// TIA Portal V16 export
// export: Created 2024-06-24T15:42:27.7485025Z, ExportSetting WithDefaults, DisplayName Totally Integrated Automation Portal, DisplayVersion V16, DisplayName TIA Portal Version Control Interface, DisplayVersion V16, DisplayName TIA Portal Openness, DisplayVersion V16, DisplayName STEP 7 Professional, DisplayVersion V16, DisplayName STEP 7 Safety, DisplayVersion V16, DisplayName WinCC Advanced, DisplayVersion V16
FUNCTION_BLOCK "FB_PickAndPlace"   // FB4, LAD
{ S7_Optimized_Access := 'TRUE' }
VERSION : 0.1
// stored: AutoNumber true, IsIECCheckEnabled false, IsRetainMemResEnabled false, MemoryReserve 100, SetENOAutomatically false, UDAEnableTagReadback false
   VAR_INPUT
      machineReady : Bool;
      movingZ : Bool;
      movingX : Bool;
      itemGrabbed : Bool;
   END_VAR
   VAR_OUTPUT
      moveX : Bool;
      moveZ : Bool;
      grabItem : Bool;
   END_VAR
   VAR_IN_OUT
      start : Bool;
      done : Bool;
   END_VAR
   VAR
      "step" : Array[0..20] of Bool;
   END_VAR
   VAR_TEMP   // added for the SCL form of the ladder/FBD networks
      _w1 : Bool;
   END_VAR
BEGIN

REGION Network 1: step0
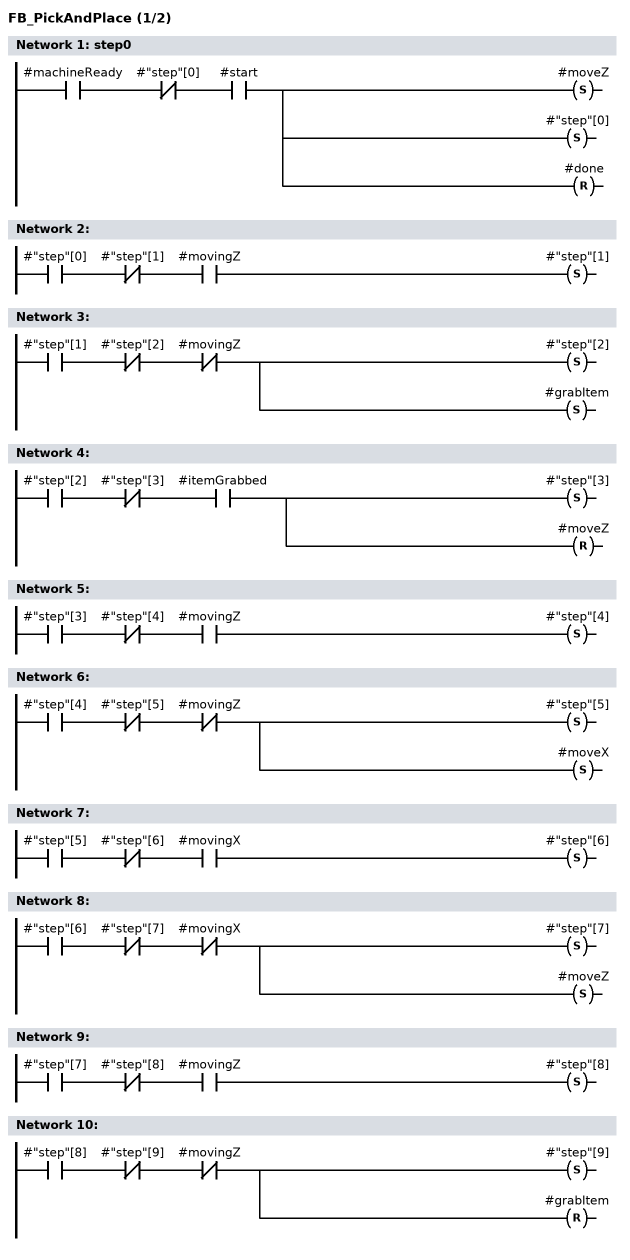
   RUNG wire#powerrail
      Contact( #machineReady )
      I_Contact( #"step"[0] )
      Contact( #start )
      wire#w1
      S_Coil( #moveZ )
   END_RUNG
   RUNG wire#w1
      S_Coil( #"step"[0] )
   END_RUNG
   RUNG wire#w1
      R_Coil( #done )
   END_RUNG
   // the same network as SCL:
   IF #machineReady AND NOT #"step"[0] AND #start THEN #moveZ := TRUE; END_IF;
   #_w1 := #machineReady AND NOT #"step"[0] AND #start;
   IF #_w1 THEN
       #"step"[0] := TRUE;
       #done := FALSE;
   END_IF;
END_REGION

REGION Network 2
   RUNG wire#powerrail
      Contact( #"step"[0] )
      I_Contact( #"step"[1] )
      Contact( #movingZ )
      S_Coil( #"step"[1] )
   END_RUNG
   // the same network as SCL:
   IF #"step"[0] AND NOT #"step"[1] AND #movingZ THEN #"step"[1] := TRUE; END_IF;
END_REGION

REGION Network 3
   RUNG wire#powerrail
      Contact( #"step"[1] )
      I_Contact( #"step"[2] )
      I_Contact( #movingZ )
      wire#w1
      S_Coil( #"step"[2] )
   END_RUNG
   RUNG wire#w1
      S_Coil( #grabItem )
   END_RUNG
   // the same network as SCL:
   #_w1 := #"step"[1] AND NOT #"step"[2] AND NOT #movingZ;
   IF #_w1 THEN
       #"step"[2] := TRUE;
       #grabItem := TRUE;
   END_IF;
END_REGION

REGION Network 4
   RUNG wire#powerrail
      Contact( #"step"[2] )
      I_Contact( #"step"[3] )
      Contact( #itemGrabbed )
      wire#w1
      S_Coil( #"step"[3] )
   END_RUNG
   RUNG wire#w1
      R_Coil( #moveZ )
   END_RUNG
   // the same network as SCL:
   #_w1 := #"step"[2] AND NOT #"step"[3] AND #itemGrabbed;
   IF #_w1 THEN
       #"step"[3] := TRUE;
       #moveZ := FALSE;
   END_IF;
END_REGION

REGION Network 5
   RUNG wire#powerrail
      Contact( #"step"[3] )
      I_Contact( #"step"[4] )
      Contact( #movingZ )
      S_Coil( #"step"[4] )
   END_RUNG
   // the same network as SCL:
   IF #"step"[3] AND NOT #"step"[4] AND #movingZ THEN #"step"[4] := TRUE; END_IF;
END_REGION

REGION Network 6
   RUNG wire#powerrail
      Contact( #"step"[4] )
      I_Contact( #"step"[5] )
      I_Contact( #movingZ )
      wire#w1
      S_Coil( #"step"[5] )
   END_RUNG
   RUNG wire#w1
      S_Coil( #moveX )
   END_RUNG
   // the same network as SCL:
   #_w1 := #"step"[4] AND NOT #"step"[5] AND NOT #movingZ;
   IF #_w1 THEN
       #"step"[5] := TRUE;
       #moveX := TRUE;
   END_IF;
END_REGION

REGION Network 7
   RUNG wire#powerrail
      Contact( #"step"[5] )
      I_Contact( #"step"[6] )
      Contact( #movingX )
      S_Coil( #"step"[6] )
   END_RUNG
   // the same network as SCL:
   IF #"step"[5] AND NOT #"step"[6] AND #movingX THEN #"step"[6] := TRUE; END_IF;
END_REGION

REGION Network 8
   RUNG wire#powerrail
      Contact( #"step"[6] )
      I_Contact( #"step"[7] )
      I_Contact( #movingX )
      wire#w1
      S_Coil( #"step"[7] )
   END_RUNG
   RUNG wire#w1
      S_Coil( #moveZ )
   END_RUNG
   // the same network as SCL:
   #_w1 := #"step"[6] AND NOT #"step"[7] AND NOT #movingX;
   IF #_w1 THEN
       #"step"[7] := TRUE;
       #moveZ := TRUE;
   END_IF;
END_REGION

REGION Network 9
   RUNG wire#powerrail
      Contact( #"step"[7] )
      I_Contact( #"step"[8] )
      Contact( #movingZ )
      S_Coil( #"step"[8] )
   END_RUNG
   // the same network as SCL:
   IF #"step"[7] AND NOT #"step"[8] AND #movingZ THEN #"step"[8] := TRUE; END_IF;
END_REGION

REGION Network 10
   RUNG wire#powerrail
      Contact( #"step"[8] )
      I_Contact( #"step"[9] )
      I_Contact( #movingZ )
      wire#w1
      S_Coil( #"step"[9] )
   END_RUNG
   RUNG wire#w1
      R_Coil( #grabItem )
   END_RUNG
   // the same network as SCL:
   #_w1 := #"step"[8] AND NOT #"step"[9] AND NOT #movingZ;
   IF #_w1 THEN
       #"step"[9] := TRUE;
       #grabItem := FALSE;
   END_IF;
END_REGION

REGION Network 11
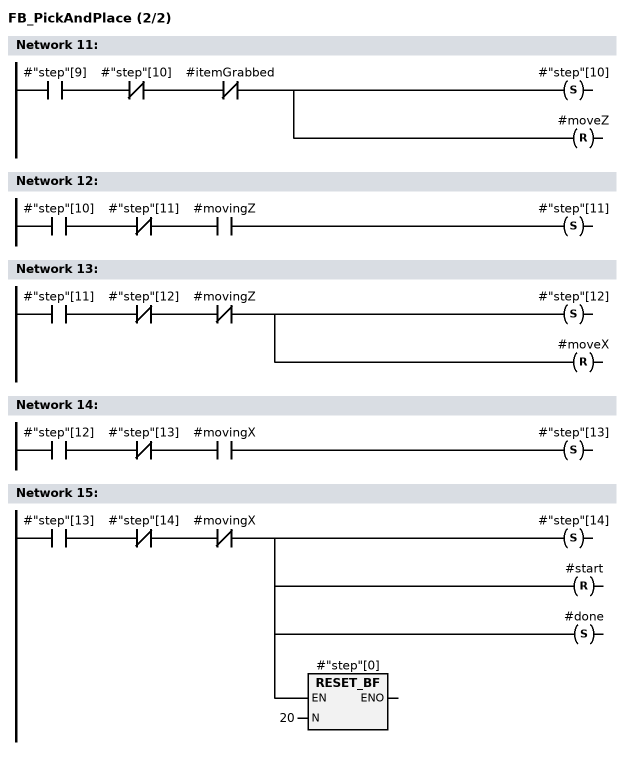
   RUNG wire#powerrail
      Contact( #"step"[9] )
      I_Contact( #"step"[10] )
      I_Contact( #itemGrabbed )
      wire#w1
      S_Coil( #"step"[10] )
   END_RUNG
   RUNG wire#w1
      R_Coil( #moveZ )
   END_RUNG
   // the same network as SCL:
   #_w1 := #"step"[9] AND NOT #"step"[10] AND NOT #itemGrabbed;
   IF #_w1 THEN
       #"step"[10] := TRUE;
       #moveZ := FALSE;
   END_IF;
END_REGION

REGION Network 12
   RUNG wire#powerrail
      Contact( #"step"[10] )
      I_Contact( #"step"[11] )
      Contact( #movingZ )
      S_Coil( #"step"[11] )
   END_RUNG
   // the same network as SCL:
   IF #"step"[10] AND NOT #"step"[11] AND #movingZ THEN #"step"[11] := TRUE; END_IF;
END_REGION

REGION Network 13
   RUNG wire#powerrail
      Contact( #"step"[11] )
      I_Contact( #"step"[12] )
      I_Contact( #movingZ )
      wire#w1
      S_Coil( #"step"[12] )
   END_RUNG
   RUNG wire#w1
      R_Coil( #moveX )
   END_RUNG
   // the same network as SCL:
   #_w1 := #"step"[11] AND NOT #"step"[12] AND NOT #movingZ;
   IF #_w1 THEN
       #"step"[12] := TRUE;
       #moveX := FALSE;
   END_IF;
END_REGION

REGION Network 14
   RUNG wire#powerrail
      Contact( #"step"[12] )
      I_Contact( #"step"[13] )
      Contact( #movingX )
      S_Coil( #"step"[13] )
   END_RUNG
   // the same network as SCL:
   IF #"step"[12] AND NOT #"step"[13] AND #movingX THEN #"step"[13] := TRUE; END_IF;
END_REGION

REGION Network 15
   // no SCL statement known for RBitfield: written as a call
   #_w1 := #"step"[13] AND NOT #"step"[14] AND NOT #movingX;
   IF #_w1 THEN
       #"step"[14] := TRUE;
       #start := FALSE;
       #done := TRUE;
       RESET_BF(operand := #"step"[0], n := 20);
   END_IF;
END_REGION
END_FUNCTION_BLOCK
